FUNCTION_BLOCK FB_PrintProfiler
VAR_INPUT
  bReset         : BOOL;
END_VAR
VAR_OUTPUT
  aProfilerData  : STRING;
  sProfilerData  : PROFILERSTRUCT;
END_VAR
VAR
  sProfiler      : T_Profiler;
END_VAR

sProfiler.stopMeasurement();
aProfilerData := sProfiler.aDataStr;
sProfilerData := sProfiler.sData;
IF bReset THEN
  bReset := FALSE;
  sProfiler.init();
END_IF
sProfiler.startMeasurement();

END_FUNCTION_BLOCK

(* stored: Version 1.1.0.1, ProductVersion 3.1.4024.3
   POU FB_PrintProfiler: Id {d3ffeeb0-0664-4b8d-8e2f-ff3d6a0fe055}, SpecialFunc None *)
